// TIA Portal V19 export
VAR_GLOBAL   // PLC tag table "tags_Open Library"
END_VAR
VAR_GLOBAL CONSTANT   // user constants
   "Modes.Auto" : Int := 1;
   "Modes.Manual" : Int := 2;
   "Modes.Independent" : Int := 10;
   "Modes.Stop" : Int := 0;
   "HMI.Status.Stopped" : Int := 0;
   "HMI.Status.Estop" : Int := 1;
   "HMI.Status.Error" : Int := 2;
   "HMI.Status.ForwardWork" : Int := 3;
   "HMI.Status.ReverseHome" : Int := 4;
   "HMI.Status.OnForwardWork" : Int := 5;
   "HMI.Status.OnReverseHome" : Int := 6;
   "IoScaling.S7Analog.Default.iRawMax" : Int := 27648;
   "IoScaling.S7Analog.Default.iRawMin" : Int := 0;
   "IoScaling.S7Analog.Default.bSwapBytes" : Bool := false;
   "IoScaling.S7Analog.+-V/mA.iRawMax" : Int := 27648;
   "IoScaling.S7Analog.+-V/mA.iRawMin" : Int := -27648;
   "IoScaling.S7Analog.Types.Default" : Int := 0;
   "IoScaling.S7Analog.Pt100.iRawMax" : Int := 8500;
   "IoScaling.S7Analog.Pt100.iRawMin" : Int := -2000;
   "IoScaling.S7Analog.Pt100.Climate.iRawMax" : Int := 13000;
   "IoScaling.S7Analog.Pt100.Climate.iRawMin" : Int := -12000;
   "IoScaling.S7Analog.Ni100.iRawMax" : Int := 2500;
   "IoScaling.S7Analog.Ni100.iRawMin" : Int := -600;
   "IoScaling.S7Analog.Ni100.Climate.iRawMax" : Int := 25000;
   "IoScaling.S7Analog.Ni100.Climate.iRawMin" : Int := -6000;
   "IoScaling.S7Analog.Types.+-V/mA" : Int := 1;
   "IoScaling.S7Analog.Types.Pt100" : Int := 2;
   "IoScaling.S7Analog.Types.Pt100.Climate" : Int := 3;
   "IoScaling.S7Analog.Types.Ni100" : Int := 4;
   "IoScaling.S7Analog.Types.Ni100.Climate" : Int := 5;
   "IoScaling.S7Analog.Pt100.rScaledMax" : Real := 850.0;
   "IoScaling.S7Analog.Pt100.rScaledMin" : Real := -200.0;
   "IoScaling.S7Analog.Pt100.Climate.rScaledMax" : Real := 130.0;
   "IoScaling.S7Analog.Pt100.Climate.rScaledMin" : Real := -120.0;
   "IoScaling.S7Analog.Ni100.rScaledMax" : Real := 250.0;
   "IoScaling.S7Analog.Ni100.rScaledMin" : Real := -60.0;
   "IoScaling.S7Analog.Ni100.Climate.rScaledMax" : Real := 250.0;
   "IoScaling.S7Analog.Ni100.Climate.rScaledMin" : Real := -60.0;
   "IoScaling.S7Analog.150Ohms.rScaledMax" : Real := 150.0;
   "IoScaling.S7Analog.150Ohms.rScaledMin" : Real := 0.0;
   "IoScaling.S7Analog.300Ohms.rScaledMax" : Real := 300.0;
   "IoScaling.S7Analog.300Ohms.rScaledMin" : Real := 0.0;
   "IoScaling.S7Analog.600Ohms.rScaledMax" : Real := 600.0;
   "IoScaling.S7Analog.600Ohms.rScaledMin" : Real := 0.0;
   "Estop.MinSetPoint" : Int := 0;
   "Estop.MaxSetPoint" : Int := 1;
   "Estop.HMISetPoint" : Int := 2;
   "Modes.PID.Inactive" : Int := 0;
   "Modes.PID.Pretuning" : Int := 1;
   "Modes.PID.FineTuning" : Int := 2;
   "Modes.PID.AutoMode" : Int := 3;
   "Modes.PID.ManualMode" : Int := 4;
   "HMI.Status.Generic1" : Int := 101;
   "HMI.Status.Generic2" : Int := 102;
   "HMI.Status.Generic3" : Int := 103;
   "HMI.Status.Generic4" : Int := 104;
   "HMI.Status.Generic5" : Int := 105;
   "HMI.Status.GenericNone" : Int := 100;
   "HMI.Status.Generic6" : Int := 106;
   "DataTypes.rMaxReal" : Real := 3.402823e38;
   "DataTypes.rMinReal" : Real := -3.402823e38;
   "DataTypes.iMaxInt" : Int := 32767;
   "DataTypes.iMinInt" : Int := -32768;
   "Handshakes.iSize" : Int := 5;
   "SoftStarter.Types.3RW30" : Int := 30;
   "SoftStarter.Types.3RW40" : Int := 40;
   "Simocode.Types.OverloadRelay" : Int := 0;
   "Simocode.Types.DirectStarter" : Int := 1;
   "Simocode.Types.ReversingStarter" : Int := 2;
   "SoftStarter.HMI.Status.RampDown" : Int := 5;
   "SoftStarter.HMI.Status.On" : Int := 4;
   "SoftStarter.HMI.Status.RampUp" : Int := 3;
   "SoftStarter.HMI.Status.EStop" : Int := 1;
   "SoftStarter.HMI.Status.Off" : Int := 0;
   "SoftStarter.HMI.Status.Error" : Int := 2;
   "FIFO.iQueueSize" : Int := 5;
   "FIFO.iQueueDisabled" : Int := -1;
   "TotalizerTimeUnits.MILLISECONDS" : Int := 0;
   "TotalizerTimeUnits.SECONDS" : Int := 1;
   "TotalizerTimeUnits.MINUTES" : Int := 2;
   "TotalizerTimeUnits.HOURS" : Int := 3;
   "TotalizerTimeUnits.DAYS" : Int := 4;
   "HMI.Status.SimulatedForwardWork" : Int := 7;
   "HMI.Status.SimulatedOnForwardWork" : Int := 9;
   "HMI.Status.SimulatedReverseHome" : Int := 8;
   "HMI.Status.SimulatedOnReverseHome" : Int := 10;
   "Ramp.Continuous" : Int := 0;
   "Ramp.Timed" : Int := 1;
END_VAR
